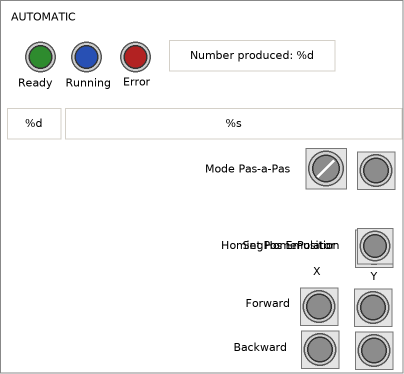
VISUALIZATION VisuAuto  // 404x374
    Label (8,2 116x30), "AUTOMATIC"
    Textfield (65,108 337x31), "%s", text variable: fbCycleAuto.fbEtape.sMess
    Lamp1 (68,39 37x36), variable: fbCycleAuto.xBusy, style: Lamp-Lamp1-Blue
    Label (59,68 59x30), "Running"
    Lamp1 (22,39 37x36), variable: fbCycleAuto.xReady, style: Lamp-Lamp1-Green
    Label (6,68 59x30), "Ready"
    Lamp1 (117,39 37x36), variable: fbCycleAuto.xError, style: Lamp-Lamp1-Red
    Label (107,67 59x30), "Error"
    Textfield (7,108 54x31), "%d", text variable: fbCycleAuto.iEtape
    Textfield (169,40 166x31), "Number produced: %d", text variable: fbCycleAuto.iNumberProduced
    RotarySwitch (305,148 42x41), variable: stParam.stStatus.xModePasAPas, behaviour: TOGGLE, style: Switch-RotarySwitch-Gray
    Label (182,154 111x30), "Mode Pas-a-Pas"
    PushSwitch (357,151 38x39), tooltip "Do next step if Pas-a-Pas is enabled", variable: fbBtn.xNextPas, invisible if: NOT stParam.stStatus.xModePasAPas, behaviour: TAP, style: Switch-PushSwitch-Gray
    Group (194,227 199x145)
        PushSwitch (161,0 38x43), variable: stIO.stIn.xSetHomePos, invisible if: fbCycleInit.iEtape<>500, behaviour: TAP, style: Switch-PushSwitch-Gray
        Label (46,4 102x29), "Set HomePosition", invisible if: fbCycleInit.iEtape<>500
        PushSwitch (106,58 38x43), variable: stIO.stIn.xJogXForward, invisible if: fbCycleInit.iEtape<>500, behaviour: TAP, style: Switch-PushSwitch-Gray
        PushSwitch (161,102 38x43), variable: stIO.stIn.xJogYBackward, invisible if: fbCycleInit.iEtape<>500, behaviour: TAP, style: Switch-PushSwitch-Gray
        PushSwitch (160,59 38x43), variable: stIO.stIn.xJogYForward, invisible if: fbCycleInit.iEtape<>500, behaviour: TAP, style: Switch-PushSwitch-Gray
        PushSwitch (107,101 38x43), variable: stIO.stIn.xJogXBackward, invisible if: fbCycleInit.iEtape<>500, behaviour: TAP, style: Switch-PushSwitch-Gray
        Label (2,62 97x29), "Forward", invisible if: fbCycleInit.iEtape<>500
        Label (0,106 96x29), "Backward", invisible if: fbCycleInit.iEtape<>500
        Label (106,30 34x29), "X", invisible if: fbCycleInit.iEtape<>500
        Label (163,35 34x29), "Y", invisible if: fbCycleInit.iEtape<>500
        Label (5,5 139x27), "HomingPos Emulator", invisible if: stParam.stStatus.xHomingDone
        PushSwitch (163,1 36x36), tooltip "Do next step if Pas-a-Pas is enabled", variable: stIO.stIn.xHomingPosReached, invisible if: stParam.stStatus.xHomingDone, behaviour: TAP, style: Switch-PushSwitch-Gray
END_VISUALIZATION

(* stored: Version 1.1.0.1, ProductVersion 3.1.4020.12
   Visu VisuAuto: Id {cb0fb055-ed28-45d9-b86b-1dc781074ad7} *)
